// TwinCAT 3 PLC project Principal
// ProgramVersion: 3.1.4023.0
// libraries:
//   Tc2_Standard, * (Beckhoff Automation GmbH)
//   Tc2_System, * (Beckhoff Automation GmbH)
//   Tc3_Module, * (Beckhoff Automation GmbH)
// project tree:
//   / PlcTask.TcTTO
//   POUs/ MAIN.TcPOU

CONFIGURATION Principal
    RESOURCE PLC ON TwinCAT3
        TASK PlcTask(INTERVAL := T#10ms, PRIORITY := 20);
        PROGRAM MAIN WITH PlcTask : MAIN;
    END_RESOURCE
END_CONFIGURATION

// ---- POUs/MAIN.TcPOU
PROGRAM MAIN
VAR
	Salida_00 AT %Q* :BOOL;
	Salida_01 AT %Q* :BOOL;
	Salida_02 AT %Q* :BOOL;
	Salida_03 AT %Q* :BOOL;
	Salida_04 AT %Q* :BOOL;
	Salida_05 AT %Q* :BOOL;
	Salida_06 AT %Q* :BOOL;
	Salida_07 AT %Q* :BOOL;
	TREN_ON :TON;
	TREN_OFF :TON;
	Contador :INT;
	RTRIGInst :R_TRIG;
	Variable_Bool :BOOL;
	Variable_Real :REAL;
	Variable_Time :TIME;
END_VAR

Variable_Time := REAL_TO_TIME(Variable_Real);
TREN_ON(IN:= NOT(TREN_OFF.Q) AND Variable_Bool, PT:= Variable_Time);
TREN_OFF(IN:= TREN_ON.Q, PT:= Variable_Time);
RTRIGInst(CLK:= TREN_ON.Q);
IF RTRIGInst.Q THEN
	Contador := Contador + 1;
END_IF;
IF Contador > 7 THEN
	Contador := 0;
END_IF;
//***************************
IF Contador = 0 THEN
	Salida_00 := TRUE;
ELSE
	Salida_00 := FALSE;
END_IF;
//***************************
IF Contador = 1 THEN
	Salida_01 := TRUE;
ELSE
	Salida_01 := FALSE;
END_IF;
//***************************
IF Contador = 2 THEN
	Salida_02 := TRUE;
ELSE
	Salida_02 := FALSE;
END_IF;
//***************************
IF Contador = 3 THEN
	Salida_03 := TRUE;
ELSE
	Salida_03 := FALSE;
END_IF;
//***************************
IF Contador = 4 THEN
	Salida_04 := TRUE;
ELSE
	Salida_04 := FALSE;
END_IF;
//***************************
IF Contador = 5 THEN
	Salida_05 := TRUE;
ELSE
	Salida_05 := FALSE;
END_IF;
//***************************
IF Contador = 6 THEN
	Salida_06 := TRUE;
ELSE
	Salida_06 := FALSE;
END_IF;
//***************************
IF Contador = 7 THEN
	Salida_07 := TRUE;
ELSE
	Salida_07 := FALSE;
END_IF;

END_PROGRAM
